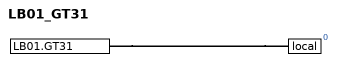
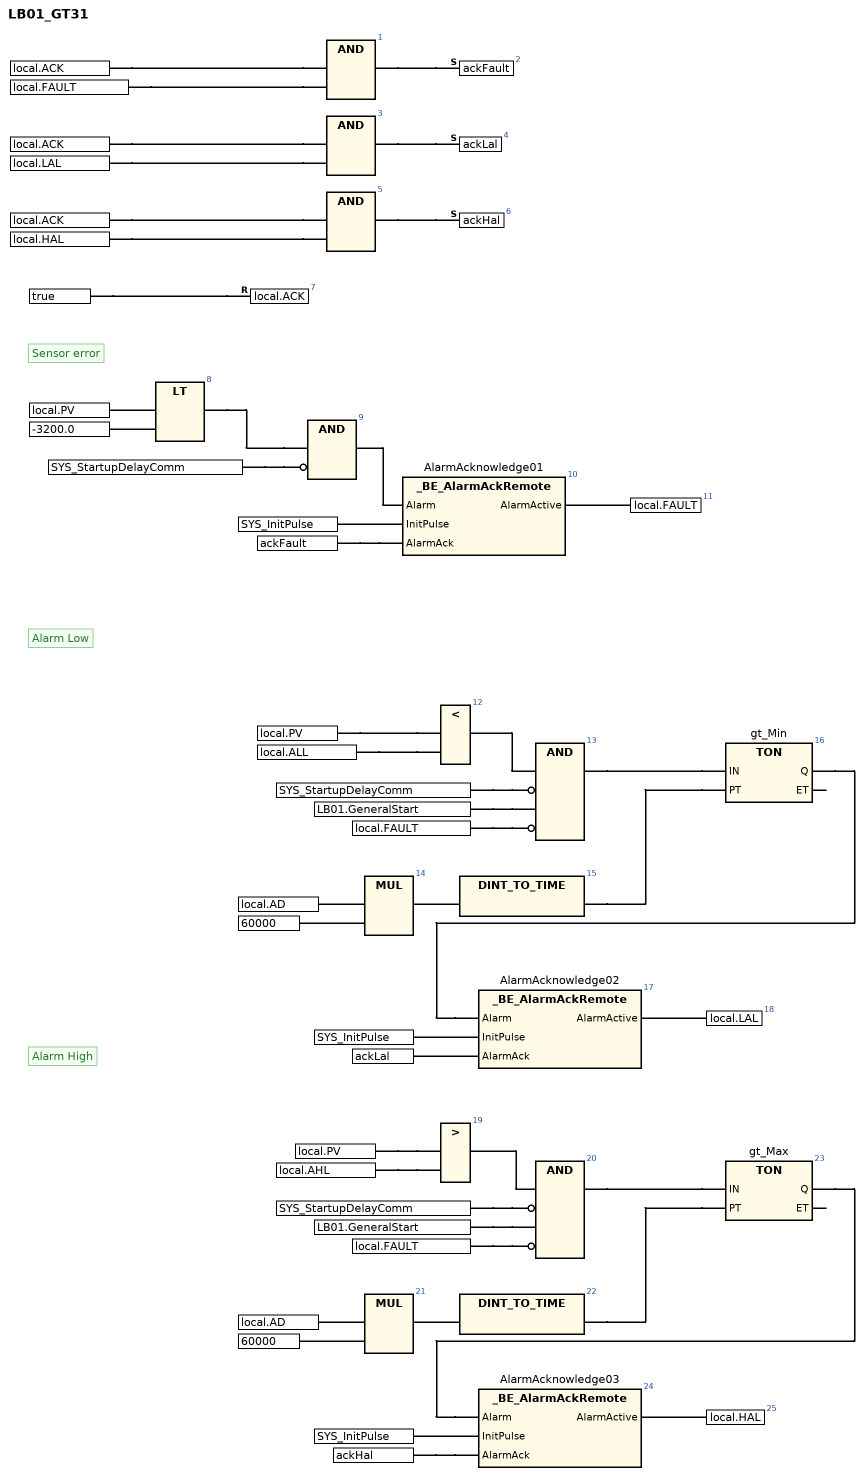
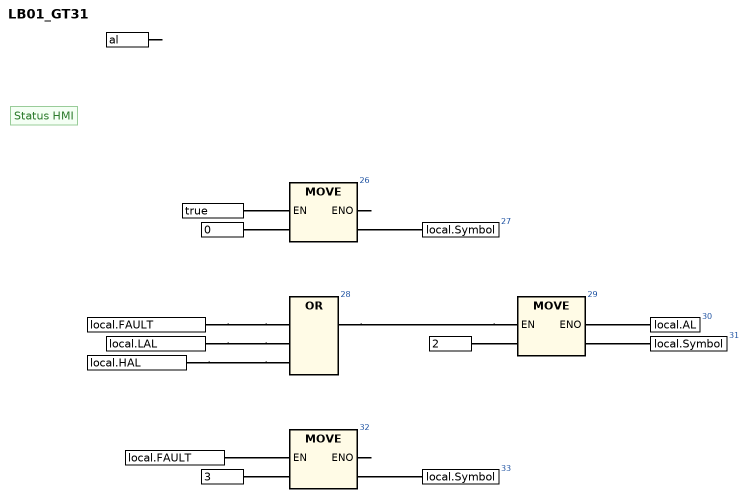
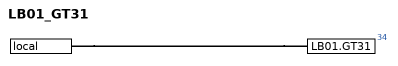
// note: 4 stored wires end on pins the file does not list and are not shown
local := LB01.GT31;
ackFault S= local.ACK AND local.FAULT;
ackLal S= local.ACK AND local.LAL;
ackHal S= local.ACK AND local.HAL;
local.ACK R= true;
// Sensor error
AlarmAcknowledge01(
    Alarm := local.PV < -3200.0 AND NOT SYS_StartupDelayComm,
    InitPulse := SYS_InitPulse,
    AlarmAck := ackFault); // _BE_AlarmAckRemote
local.FAULT := AlarmAcknowledge01.AlarmActive;
// Alarm Low
gt_Min(IN := local.PV < local.ALL AND NOT SYS_StartupDelayComm AND LB01.GeneralStart AND NOT local.FAULT, PT := DINT_TO_TIME(local.AD * 60000)); // TON
AlarmAcknowledge02(Alarm := gt_Min.Q, InitPulse := SYS_InitPulse, AlarmAck := ackLal); // _BE_AlarmAckRemote
local.LAL := AlarmAcknowledge02.AlarmActive;
// Alarm High
gt_Max(IN := local.PV > local.AHL AND NOT SYS_StartupDelayComm AND LB01.GeneralStart AND NOT local.FAULT, PT := DINT_TO_TIME(local.AD * 60000)); // TON
AlarmAcknowledge03(Alarm := gt_Max.Q, InitPulse := SYS_InitPulse, AlarmAck := ackHal); // _BE_AlarmAckRemote
local.HAL := AlarmAcknowledge03.AlarmActive;
// Status HMI
IF true THEN _w1 := 0; END_IF
local.Symbol := _w1;
_w2 := local.FAULT OR local.LAL OR local.HAL;
IF _w2 THEN _w3 := 2; END_IF
local.AL := _w2;
local.Symbol := _w3;
IF local.FAULT THEN _w4 := 3; END_IF
local.Symbol := _w4;
LB01.GT31 := local;
// al: input not connected

END_PROGRAM

// Device/AREA1/B001/LB01/Sensor/Temperature/GT21/LB01_Cascade_ExtractControl
PROGRAM LB01_Cascade_ExtractControl
VAR
END_VAR
VAR // added by the converter: edge detectors and wires of the graphical bodies
    _w1 : ANY;
END_VAR

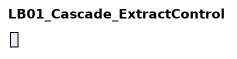
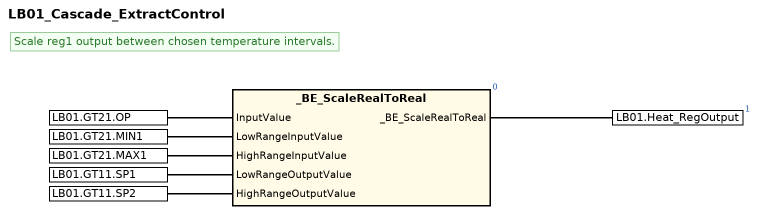
// Scale reg1 output between chosen temperature intervals.
_w1 := _BE_ScaleRealToReal(InputValue := LB01.GT21.OP, LowRangeInputValue := LB01.GT21.MIN1, HighRangeInputValue := LB01.GT21.MAX1, LowRangeOutputValue := LB01.GT11.SP1, HighRangeOutputValue := LB01.GT11.SP2);
LB01.Heat_RegOutput := _w1;

END_PROGRAM

// Device/AREA1/B001/LB01/Sensor/Pressure/GP91/LB01_GP91
PROGRAM LB01_GP91
VAR
	local:strSensor10_HeatExchanger_Pressure;
	AlarmAcknowledge01: _BE_AlarmAckRemote;
END_VAR
VAR // added by the converter: edge detectors and wires of the graphical bodies
    _w1, _w3 : ANY;
    _w2 : BOOL;
END_VAR

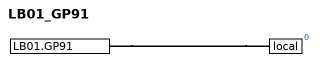
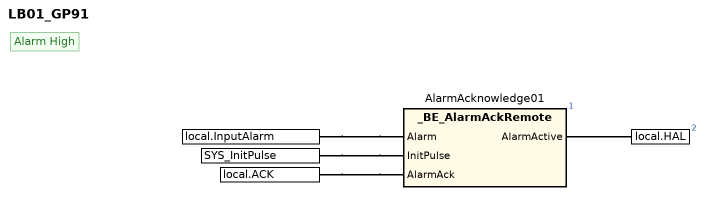
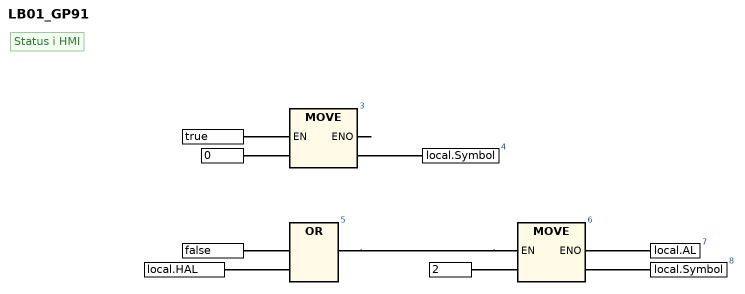
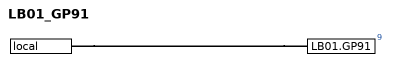
local := LB01.GP91;
// Alarm High
AlarmAcknowledge01(Alarm := local.InputAlarm, InitPulse := SYS_InitPulse, AlarmAck := local.ACK); // _BE_AlarmAckRemote
local.HAL := AlarmAcknowledge01.AlarmActive;
// Status i HMI
IF true THEN _w1 := 0; END_IF
local.Symbol := _w1;
_w2 := false OR local.HAL;
IF _w2 THEN _w3 := 2; END_IF
local.AL := _w2;
local.Symbol := _w3;
LB01.GP91 := local;

END_PROGRAM

// Device/AREA1/B001/LB01/Sensor/Temperature/GT21/LB01_GT21_Control
PROGRAM LB01_GT21_Control
VAR
	local:strSensor2_Regulator;
	gt_Min: TON;
	gt_Max: TON;
	reset_en: RS;
	FbRegulator: _BE_Regulator;
	ackFault: BOOL;
	ackLal: BOOL;
	ackHal: BOOL;
	AlarmAcknowledge01: _BE_AlarmAckRemote;
	AlarmAcknowledge02: _BE_AlarmAckRemote;
	AlarmAcknowledge03: _BE_AlarmAckRemote;
END_VAR
VAR // added by the converter: edge detectors and wires of the graphical bodies
    _w1, _w4, _w5, _w6, _w8, _w9 : ANY;
    _w2, _w3, _w7 : BOOL;
END_VAR

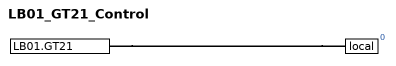
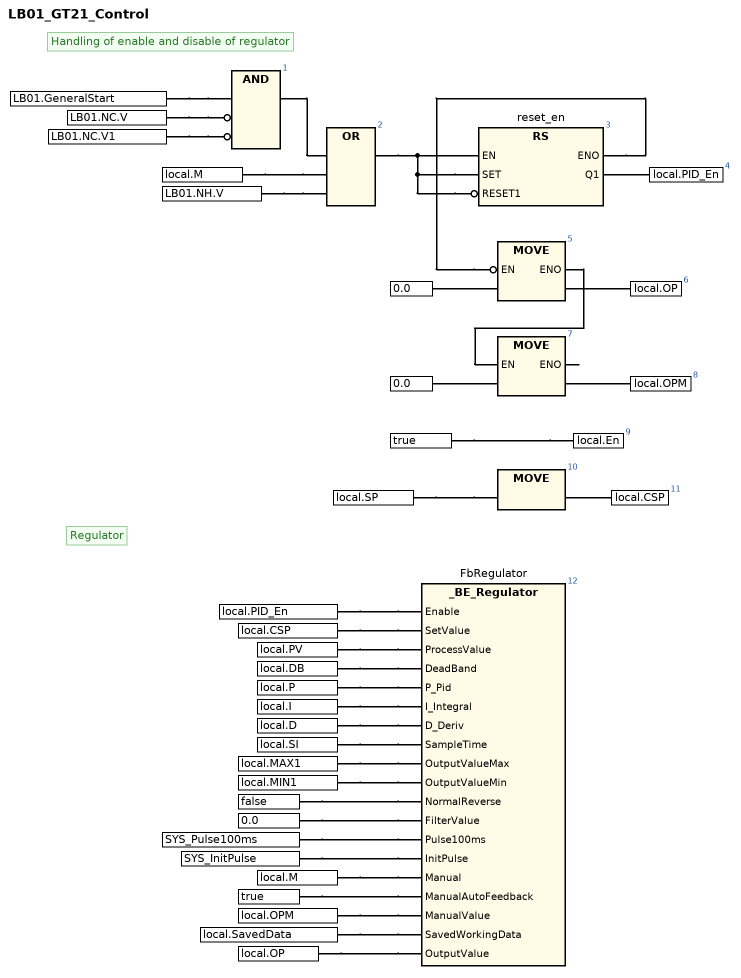
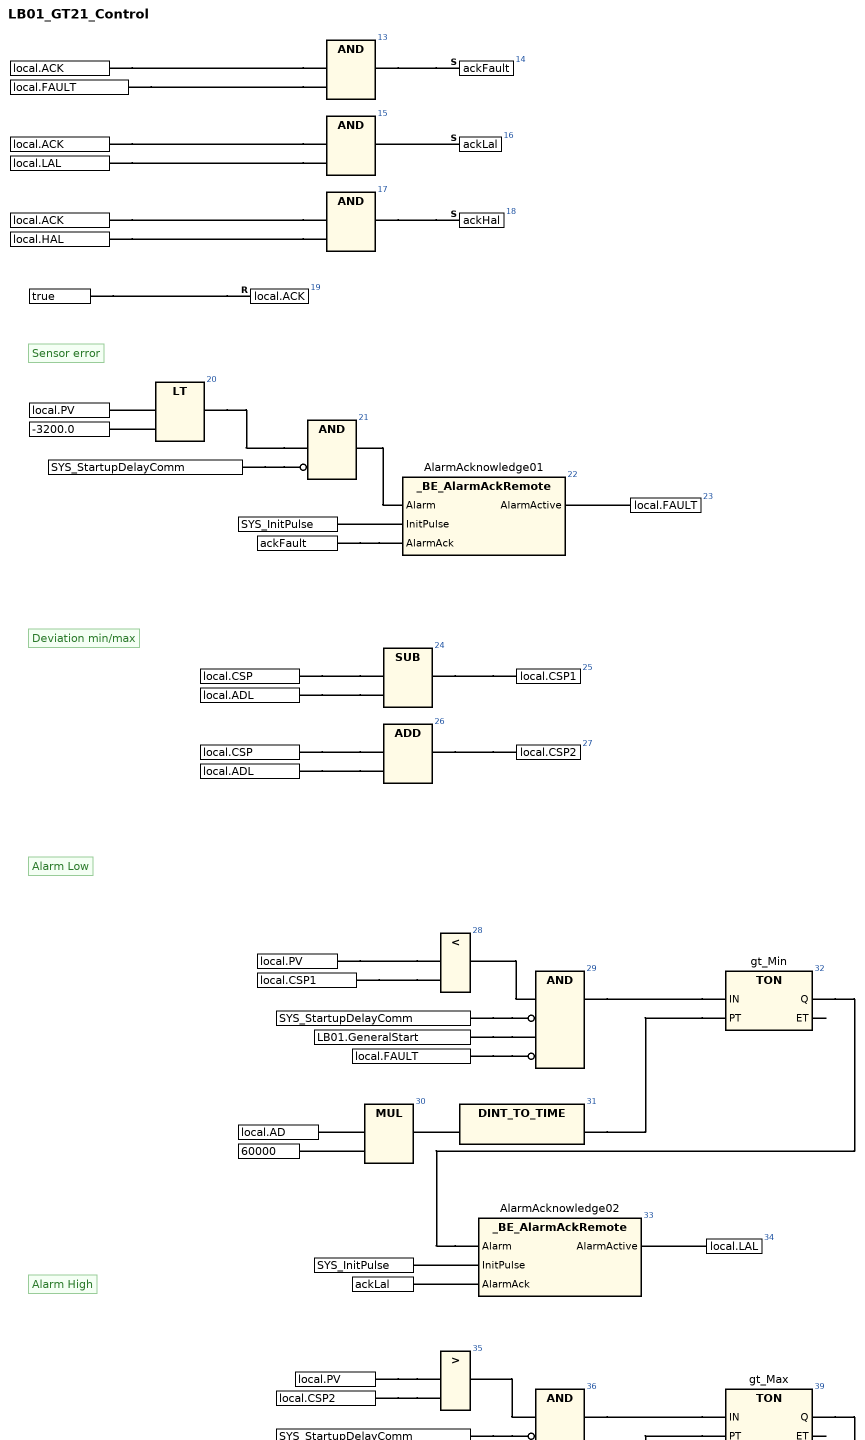
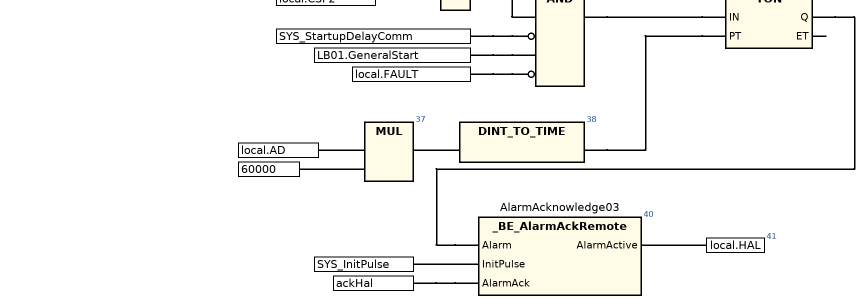
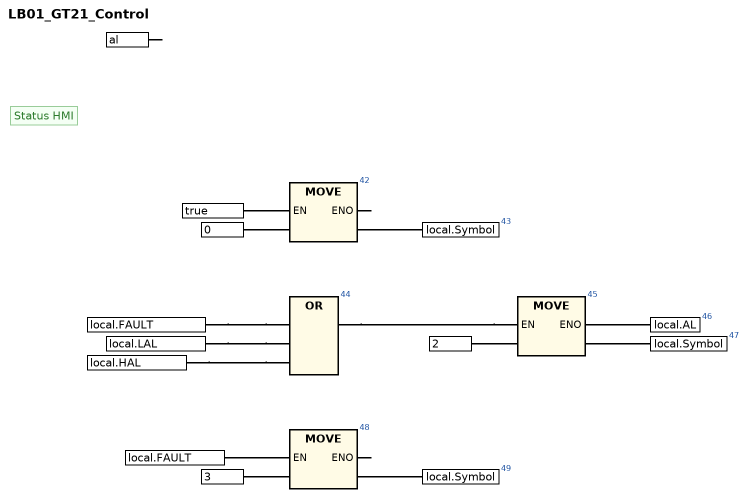
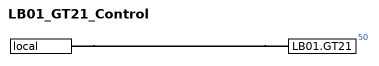
local := LB01.GT21;
// Handling of enable and disable of regulator
_w1 := LB01.GeneralStart AND NOT LB01.NC.V AND NOT LB01.NC.V1 OR local.M OR LB01.NH.V;
_w2 := _w1;
IF _w2 THEN
    reset_en(SET := _w1, RESET1 := NOT _w1); // RS
END_IF
local.PID_En := reset_en.Q1;
_w3 := NOT _w2;
IF _w3 THEN _w4 := 0.0; END_IF
local.OP := _w4;
IF _w3 THEN _w5 := 0.0; END_IF
local.OPM := _w5;
local.En := true;
local.CSP := local.SP;
// Regulator
FbRegulator(
    Enable := local.PID_En,
    SetValue := local.CSP,
    ProcessValue := local.PV,
    DeadBand := local.DB,
    P_Pid := local.P,
    I_Integral := local.I,
    D_Deriv := local.D,
    SampleTime := local.SI,
    OutputValueMax := local.MAX1,
    OutputValueMin := local.MIN1,
    NormalReverse := false,
    FilterValue := 0.0,
    Pulse100ms := SYS_Pulse100ms,
    InitPulse := SYS_InitPulse,
    Manual := local.M,
    ManualAutoFeedback := true,
    ManualValue := local.OPM,
    SavedWorkingData := local.SavedData,
    OutputValue := local.OP); // _BE_Regulator
ackFault S= local.ACK AND local.FAULT;
ackLal S= local.ACK AND local.LAL;
ackHal S= local.ACK AND local.HAL;
local.ACK R= true;
// Sensor error
AlarmAcknowledge01(
    Alarm := local.PV < -3200.0 AND NOT SYS_StartupDelayComm,
    InitPulse := SYS_InitPulse,
    AlarmAck := ackFault); // _BE_AlarmAckRemote
local.FAULT := AlarmAcknowledge01.AlarmActive;
// Deviation min/max
local.CSP1 := local.CSP - local.ADL;
local.CSP2 := local.CSP + local.ADL;
// Alarm Low
gt_Min(IN := local.PV < local.CSP1 AND NOT SYS_StartupDelayComm AND LB01.GeneralStart AND NOT local.FAULT, PT := DINT_TO_TIME(local.AD * 60000)); // TON
AlarmAcknowledge02(Alarm := gt_Min.Q, InitPulse := SYS_InitPulse, AlarmAck := ackLal); // _BE_AlarmAckRemote
local.LAL := AlarmAcknowledge02.AlarmActive;
// Alarm High
gt_Max(IN := local.PV > local.CSP2 AND NOT SYS_StartupDelayComm AND LB01.GeneralStart AND NOT local.FAULT, PT := DINT_TO_TIME(local.AD * 60000)); // TON
AlarmAcknowledge03(Alarm := gt_Max.Q, InitPulse := SYS_InitPulse, AlarmAck := ackHal); // _BE_AlarmAckRemote
local.HAL := AlarmAcknowledge03.AlarmActive;
// Status HMI
IF true THEN _w6 := 0; END_IF
local.Symbol := _w6;
_w7 := local.FAULT OR local.LAL OR local.HAL;
IF _w7 THEN _w8 := 2; END_IF
local.AL := _w7;
local.Symbol := _w8;
IF local.FAULT THEN _w9 := 3; END_IF
local.Symbol := _w9;
LB01.GT21 := local;
// al: input not connected

END_PROGRAM

// Device/AREA1/B001/LB01/Damper/ST11/LB01_ST11_Analog
PROGRAM LB01_ST11_Analog
VAR
	local:strDamper_Analog;
	FbPulse: R_TRIG;
	delayST11: TON;
	sp1: DINT;
	operating: BOOL;
	nh_v: BOOL;
END_VAR
VAR // added by the converter: edge detectors and wires of the graphical bodies
    _w1, _w2, _w3 : ANY;
END_VAR

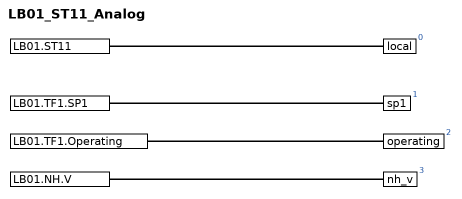
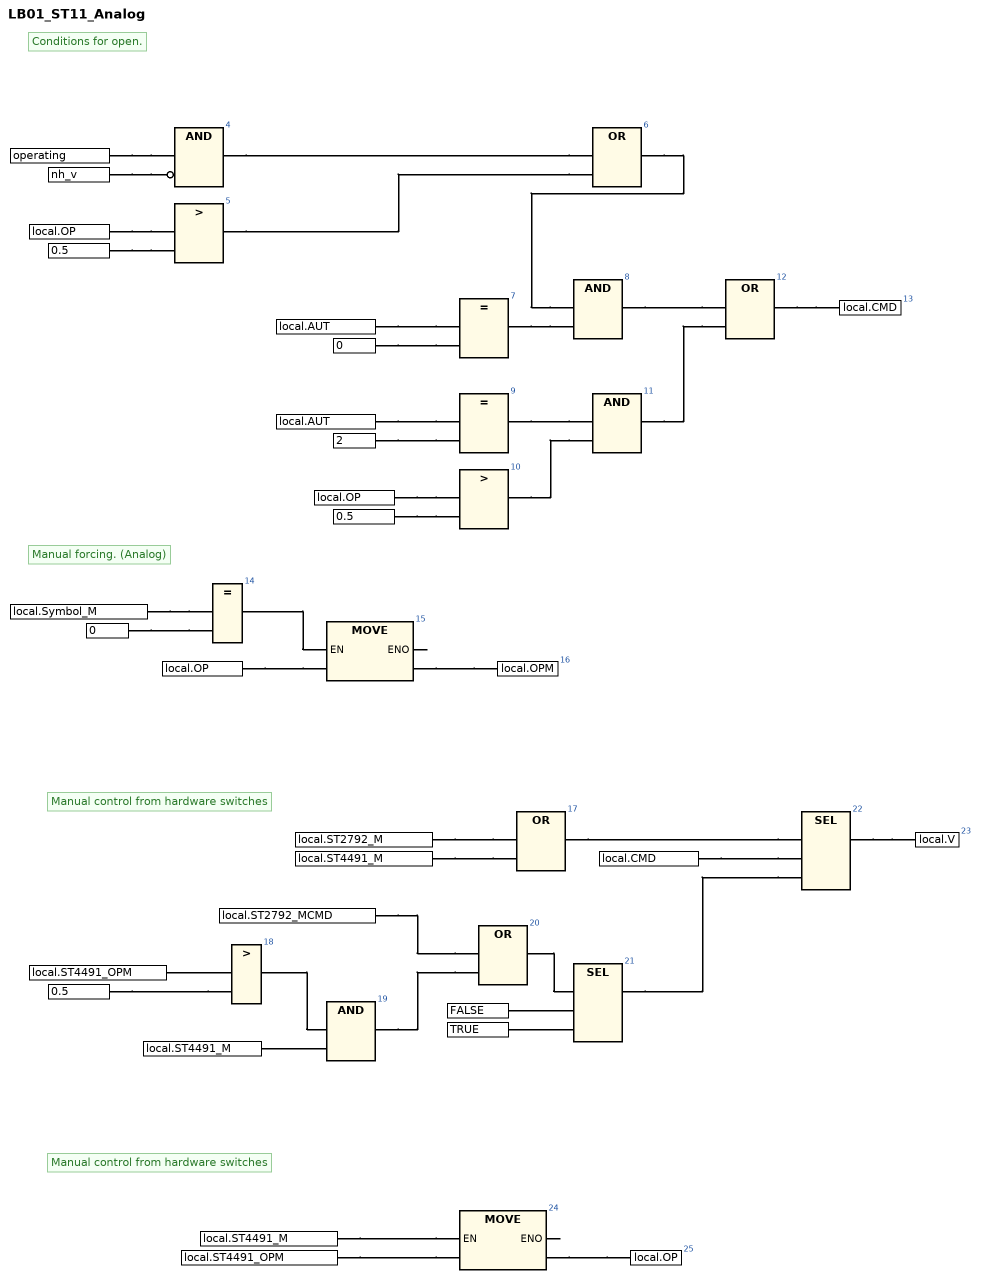
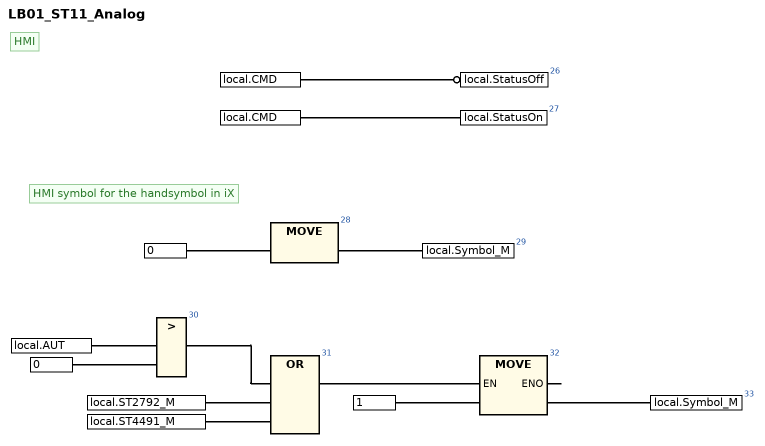
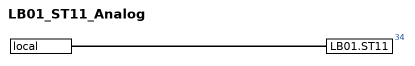
local := LB01.ST11;
sp1 := LB01.TF1.SP1;
operating := LB01.TF1.Operating;
nh_v := LB01.NH.V;
// Conditions for open.
local.CMD := (operating AND NOT nh_v OR local.OP > 0.5) AND local.AUT = 0 OR local.AUT = 2 AND local.OP > 0.5;
// Manual forcing. (Analog)
IF local.Symbol_M = 0 THEN _w1 := local.OP; END_IF
local.OPM := _w1;
// Manual control from hardware switches
local.V := SEL(local.ST2792_M OR local.ST4491_M, local.CMD, SEL(local.ST2792_MCMD OR local.ST4491_OPM > 0.5 AND local.ST4491_M, FALSE, TRUE));
// Manual control from hardware switches
IF local.ST4491_M THEN _w2 := local.ST4491_OPM; END_IF
local.OP := _w2;
// HMI
local.StatusOff := NOT local.CMD;
local.StatusOn := local.CMD;
// HMI symbol for the handsymbol in iX
local.Symbol_M := 0;
IF local.AUT > 0 OR local.ST2792_M OR local.ST4491_M THEN _w3 := 1; END_IF
local.Symbol_M := _w3;
LB01.ST11 := local;

END_PROGRAM

// Device/AREA1/B001/LB01/Damper/ST21/LB01_ST21_Analog
PROGRAM LB01_ST21_Analog
VAR
	local:strDamper_Analog;
	FbPulse: R_TRIG;
	delayST11: TON;
	sp1: DINT;
	operating: BOOL;
	nh_v: BOOL;
END_VAR
VAR // added by the converter: edge detectors and wires of the graphical bodies
    _w1, _w2, _w3 : ANY;
END_VAR

